SUBAPPLICATION OPC_PUB_FIO (* Subapplication Type *)
  (* Standard: 61499-2 *)
  (* Version 1.0, 2022-03-11, Maximilian Scharf *)
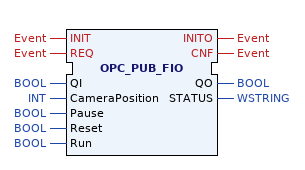
  EVENT_INPUT
    INIT;
    REQ;
  END_EVENT
  EVENT_OUTPUT
    INITO;
    CNF;
  END_EVENT
  VAR_INPUT
    QI : BOOL;
    CameraPosition : INT;
    Pause : BOOL;
    Reset : BOOL;
    Run : BOOL;
  END_VAR
  VAR_OUTPUT
    QO : BOOL;
    STATUS : WSTRING;
  END_VAR
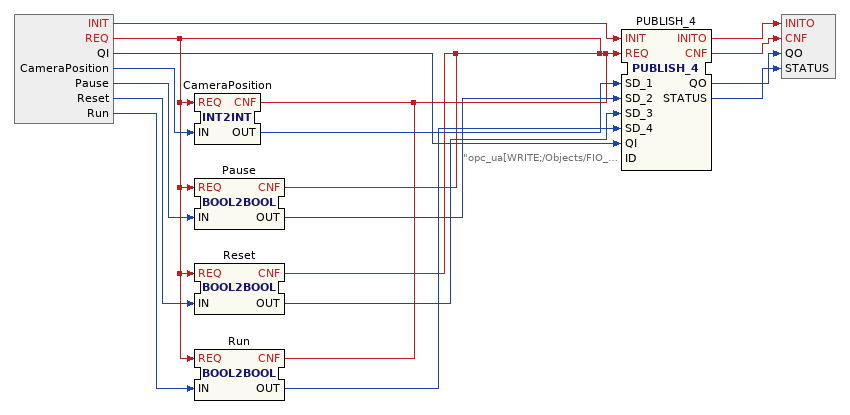
  FBS
    PUBLISH_4 : PUBLISH_4(ID := "opc_ua[WRITE;/Objects/FIO_Q_CameraPosition, 1:s=FIO_Q_CameraPosition;/Objects/FIO_Q_Pause, 1:s=FIO_Q_Pause;/Objects/FIO_Q_Reset, 1:s=FIO_Q_Reset;/Objects/FIO_Q_Run, 1:s=FIO_Q_Run]");
    CameraPosition : INT2INT;
    Pause : BOOL2BOOL;
    Reset : BOOL2BOOL;
    Run : BOOL2BOOL;
  END_FBS
  EVENT_CONNECTIONS
    INIT TO PUBLISH_4.INIT;
    REQ TO PUBLISH_4.REQ;
    PUBLISH_4.INITO TO INITO;
    PUBLISH_4.CNF TO CNF;
    CameraPosition.CNF TO PUBLISH_4.REQ;
    REQ TO CameraPosition.REQ;
    REQ TO Pause.REQ;
    REQ TO Reset.REQ;
    REQ TO Run.REQ;
    Pause.CNF TO PUBLISH_4.REQ;
    Reset.CNF TO PUBLISH_4.REQ;
    Run.CNF TO PUBLISH_4.REQ;
  END_CONNECTIONS
  DATA_CONNECTIONS
    PUBLISH_4.QO TO QO;
    PUBLISH_4.STATUS TO STATUS;
    CameraPosition.OUT TO PUBLISH_4.SD_1;
    CameraPosition TO CameraPosition.IN;
    Pause TO Pause.IN;
    Reset TO Reset.IN;
    Run TO Run.IN;
    Pause.OUT TO PUBLISH_4.SD_2;
    Reset.OUT TO PUBLISH_4.SD_3;
    Run.OUT TO PUBLISH_4.SD_4;
    QI TO PUBLISH_4.QI;
  END_CONNECTIONS
END_SUBAPPLICATION
